(* PLC project  *)

CONFIGURATION Empty_Module_26
END_CONFIGURATION
